ABB RAPID module: 001E1CDD

MODULE Module1
    CONST robtarget AboveDuster:=[[743.879676977,-800.509897995,1300.071035327],[0.000000006,0.382683505,0.923879502,0.000000013],[-1,0,-2,0],[9E+09,9E+09,9E+09,9E+09,9E+09,9E+09]];
    CONST robtarget Duster:=[[743.879739272,-800.509937926,866.646225387],[0,0.382683433,0.923879532,0],[-1,0,-2,0],[9E+09,9E+09,9E+09,9E+09,9E+09,9E+09]];
ENDMODULE
